Universal Robots PolyScope program: pick_up_bottle_cups_xijun.urp

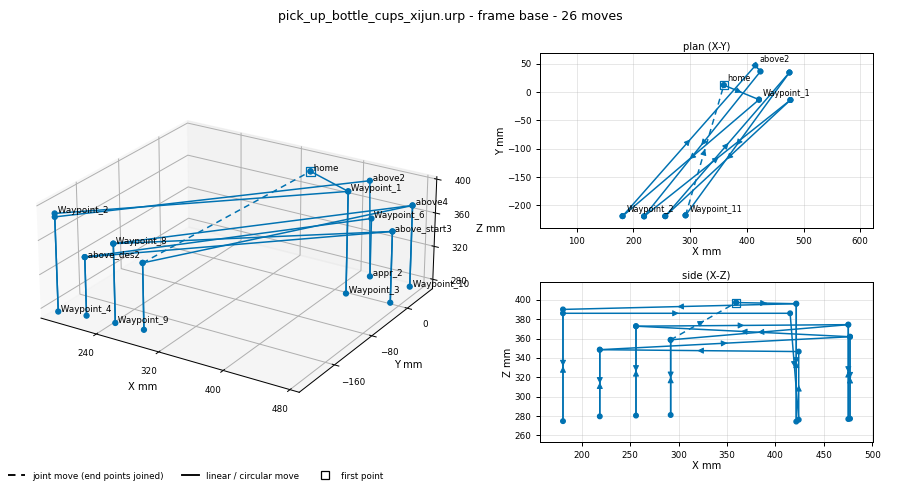
[picture p0: tool path of pick_up_bottle_cups_xijun.urp in frame base, 26 of 26 moves have a stored position in this frame; points joined in program order, loops and branches not executed]
Program pick_up_bottle_cups_xijun (installation=default directory=/programs/TM1326 createdIn=5.11.9.1010452 lastSavedIn=5.11.9.1010452 robotSerialNumber=20225200364)
Calibrated DH parameters: a=[0.00002, -0.569483, -0.54992, -0.00001, -0.000036, 0]; d=[0.180894, -146.691669, 192.918669, -46.053088, 0.119778, 0.115602]; alpha=[1.571425, -0.001534, 0.003359, 1.568739, -1.571477, 0]; deltaTheta=[0, 0.376258, -0.101074, -0.275185, -0.000002, 0]
Robot Program (runOnlyOnce=false)
  MoveL speed 250 mm/s, acceleration 1200 mm/s^2 (useActiveTCP=true) feature=Base
    Waypoint home: TCP in base x=359.452 y=12.315 z=397.104 mm, rx=2.2285 ry=-2.2071 rz=-0.0059 rad; joints [30.896, -83.989, -125.155, -241.227, -90.276, -149.493] deg
    URCap RG Grip (OnRobot, OnRobot A/S) dataModel(rg-target-force=3.0, rg-target-width=0.04)
    Waypoint Waypoint_1: TCP in base x=421.49 y=-13.305 z=395.907 mm, rx=2.2286 ry=-2.2069 rz=-0.0057 rad; joints [22.574, -90.728, -118.938, -240.723, -90.215, -157.82] deg
    Waypoint Waypoint_3: TCP in base x=421.478 y=-13.325 z=274.291 mm, rx=2.2285 ry=-2.207 rz=-0.0058 rad; joints [22.578, -98.774, -125.27, -226.345, -90.196, -157.773] deg
    URCap RG Grip (OnRobot, OnRobot A/S) dataModel(rg-target-force=3.0, rg-target-width=0.032, Variable(key=on_return, variable(name=on_return)))
    Waypoint Waypoint_1: TCP in base x=421.49 y=-13.305 z=395.907 mm, rx=2.2286 ry=-2.2069 rz=-0.0057 rad; joints [22.574, -90.728, -118.938, -240.723, -90.215, -157.82] deg
  MoveL speed 250 mm/s, acceleration 1200 mm/s^2 (useActiveTCP=true) feature=Base
    Waypoint Waypoint_2: TCP in base x=180.759 y=-218.871 z=390.033 mm, rx=2.2285 ry=-2.2071 rz=-0.0056 rad; joints [-12.493, -74.746, -133.128, -242.49, -90.011, -192.888] deg
    Waypoint Waypoint_4: TCP in base x=180.762 y=-218.866 z=274.724 mm, rx=2.2286 ry=-2.2071 rz=-0.0056 rad; joints [-12.472, -84.035, -140.484, -225.842, -89.991, -192.82] deg
    URCap RG Grip (OnRobot, OnRobot A/S) dataModel(rg-target-force=3.0, rg-target-width=0.04)
    Waypoint Waypoint_5: TCP in base x=180.743 y=-218.865 z=386.038 mm, rx=2.2285 ry=-2.2072 rz=-0.0057 rad; joints [-12.494, -74.985, -133.419, -241.959, -90.015, -192.885] deg
    Waypoint above2: TCP in base x=415.149 y=46.9 z=386.038 mm, rx=2.2285 ry=-2.2072 rz=-0.0057 rad; joints [31.056, -90.859, -119.944, -239.562, -90.265, -149.325] deg
    Waypoint appr_2: TCP in base x=424.025 y=36.453 z=276.203 mm, rx=2.2284 ry=-2.2072 rz=-0.0058 rad; joints [29.053, -98.973, -124.755, -226.644, -90.235, -151.29] deg
    URCap RG Grip (OnRobot, OnRobot A/S) dataModel(rg-target-force=3.0, rg-target-width=0.032, rg-depth-compensation-enabled=true)
    Waypoint Waypoint_6: TCP in base x=424.033 y=36.49 z=346.54 mm, rx=2.2286 ry=-2.2071 rz=-0.0057 rad; joints [29.054, -93.982, -121.38, -235.01, -90.246, -151.319] deg
    Waypoint above_des2: TCP in base x=218.753 y=-219.185 z=348.476 mm, rx=2.2288 ry=-2.207 rz=-0.0056 rad; joints [-10.742, -81.013, -133.376, -235.974, -90.018, -191.127] deg
    Waypoint Waypoint_7: TCP in base x=218.74 y=-219.199 z=279.671 mm, rx=2.2287 ry=-2.2071 rz=-0.0056 rad; joints [-10.736, -86.8, -137.356, -226.205, -90.004, -191.089] deg
    URCap RG Grip (OnRobot, OnRobot A/S) dataModel(rg-target-width=0.04, rg-target-force=3.0)
    Waypoint above_des2: TCP in base x=218.753 y=-219.185 z=348.476 mm, rx=2.2288 ry=-2.207 rz=-0.0056 rad; joints [-10.742, -81.013, -133.376, -235.974, -90.018, -191.127] deg
  MoveL speed 250 mm/s, acceleration 1200 mm/s^2 (useActiveTCP=true) feature=Base
    Waypoint above_start3: TCP in base x=476.97 y=-13.898 z=361.841 mm, rx=2.2288 ry=-2.2071 rz=-0.0056 rad; joints [19.73, -97.982, -114.986, -237.408, -90.189, -160.654] deg
    Waypoint pick3: TCP in base x=476.97 y=-13.876 z=277.291 mm, rx=2.2288 ry=-2.207 rz=-0.0056 rad; joints [19.735, -103.395, -118.927, -228.055, -90.176, -160.625] deg
    URCap RG Grip (OnRobot, OnRobot A/S) dataModel(rg-target-force=3.0, rg-target-width=0.032, rg-depth-compensation-enabled=true)
    Waypoint above_start3: TCP in base x=476.97 y=-13.898 z=361.841 mm, rx=2.2288 ry=-2.2071 rz=-0.0056 rad; joints [19.73, -97.982, -114.986, -237.408, -90.189, -160.654] deg
    Waypoint Waypoint_8: TCP in base x=256.105 y=-218.931 z=372.723 mm, rx=2.2288 ry=-2.207 rz=-0.0056 rad; joints [-9.327, -82.748, -129.052, -238.564, -90.027, -189.719] deg
    Waypoint Waypoint_9: TCP in base x=256.108 y=-218.932 z=280.484 mm, rx=2.2288 ry=-2.207 rz=-0.0056 rad; joints [-9.316, -89.85, -134.326, -226.191, -90.007, -189.673] deg
    URCap RG Grip (OnRobot, OnRobot A/S) dataModel(rg-target-width=0.04, rg-target-force=3.0)
    Waypoint Waypoint_8: TCP in base x=256.105 y=-218.931 z=372.723 mm, rx=2.2288 ry=-2.207 rz=-0.0056 rad; joints [-9.327, -82.748, -129.052, -238.564, -90.027, -189.719] deg
  MoveL speed 250 mm/s, acceleration 1200 mm/s^2 (useActiveTCP=true) feature=Base
    Waypoint above4: TCP in base x=475.18 y=34.611 z=374.298 mm, rx=-2.241 ry=2.2017 rz=0 rad; joints [25.615, -97.125, -114.423, -238.483, -90.128, -155.223] deg
    Waypoint Waypoint_10: TCP in base x=475.185 y=34.616 z=276.924 mm, rx=2.2409 ry=-2.2017 rz=0 rad; joints [25.619, -103.25, -119.073, -227.714, -90.111, -155.191] deg
    URCap RG Grip (OnRobot, OnRobot A/S) dataModel(rg-target-force=3.0, rg-target-width=0.032, rg-depth-compensation-enabled=true)
    Waypoint above4: TCP in base x=475.18 y=34.611 z=374.298 mm, rx=-2.241 ry=2.2017 rz=0 rad; joints [25.615, -97.125, -114.423, -238.483, -90.128, -155.223] deg
    Waypoint Waypoint_11: TCP in base x=291.878 y=-217.433 z=358.65 mm, rx=2.241 ry=-2.2017 rz=0.0001 rad; joints [-8.071, -86.671, -127.185, -236.174, -90.133, -188.905] deg
    Waypoint Waypoint_12: TCP in base x=291.892 y=-217.428 z=281.087 mm, rx=2.241 ry=-2.2017 rz=0.0001 rad; joints [-8.062, -92.546, -131.363, -226.122, -90.116, -188.869] deg
    URCap RG Grip (OnRobot, OnRobot A/S) dataModel(rg-target-width=0.04, rg-target-force=3.0)
    Waypoint Waypoint_11: TCP in base x=291.878 y=-217.433 z=358.65 mm, rx=2.241 ry=-2.2017 rz=0.0001 rad; joints [-8.071, -86.671, -127.185, -236.174, -90.133, -188.905] deg
  MoveJ speed 60 deg/s, acceleration 80 deg/s^2 (useActiveTCP=true) feature=Base
    Waypoint home: TCP in base x=359.452 y=12.315 z=397.104 mm, rx=2.2285 ry=-2.2071 rz=-0.0059 rad; joints [30.896, -83.989, -125.155, -241.227, -90.276, -149.493] deg
    Halt
